Fanuc KAREL source: ko00076.KL

-- PROVISIONAL review KL for V940-1; original PC SHA256 d94709dd2466d7e425af88cd5902512d4c828994e91d038c4d183e46b906940f
-- Incomplete behavior may be omitted. Consult companion uncertainty JSON. Do not deploy.
PROGRAM KO00076
%NOLOCKGROUP
BEGIN
  -- V9_ZERO_TABLE_METADATA_HINT layout=0002_ascii; no indexed target words; source/name/runtime held
  -- UNRESOLVED_PC offsets 5-12; opcodes 9D,23
  -- UNRESOLVED_PC offsets 17-66; opcodes 27,22,1C,27,49,7E,AD,22,31,7E,4A
  -- UNRESOLVED_PC offsets 71-75; opcodes 7F
END KO00076
